// TIA Portal V19 export
DATA_BLOCK "HmiInterface"   // DB60
// stored: Access Published, MemoryReserve 100, Namespace Unit2.EM1
   VAR
      em : "LAF_typeEmInterface";
      jobs : "LAF_typeJobsInterface";
      sequence : "LAF_typeSequenceInterface";
      cm1Vfd205 : "LEXCHANGETRAY_typeRollerVfdInterface";
      cm2SingalTM : "LEXCHANGETRAY_typeRollerIoSignalInterface";
      em1Parameters : "LAF_typeRollerEm1ParametersInterface";
   END_VAR
BEGIN
END_DATA_BLOCK
